// TwinCAT 3 PLC project Untitled1
// ProgramVersion: 3.1.4023.0
// libraries:
//   EfficientIO Communicator, * (EfficientIO)
//   EfficientIO Energy Basic, * (EfficientIO)
//   EfficientIO ModbusTCP, * (EfficientIO)
//   Lynus HTTP Functions, * (Lynus AG)
//   Lynus Standards, * (EfficientIO)
//   Tc2_Standard, * (Beckhoff Automation GmbH)
//   Tc2_System, * (Beckhoff Automation GmbH)
//   Tc2_Utilities, * (Beckhoff Automation GmbH)
//   Tc3_Module, * (Beckhoff Automation GmbH)
// project tree:
//   / Com.TcTTO, Lynus.TcTTO, PlcTask.TcTTO
//   DUTs/ struct_ADS_Auhofcenter.TcDUT
//   FBs/ FB_SPOpt_Monitoring_extTime.TcPOU
//   POUs/ MAIN.TcPOU, prgCom.TcPOU, prgLynus.TcPOU, prgPV.TcPOU
// real-time tasks:
//   TASK PlcTask: cycle T#10ms, priority 10, ADS port 350
//   TASK Com: cycle T#20ms, priority 14, ADS port 352
//   TASK Lynus: cycle T#5ms, priority 6, ADS port 351
//   TASK Riverside_Fast: cycle T#5ms, priority 8, ADS port 353
//   TASK Riverside_Middle: cycle T#20ms, priority 12, ADS port 354

CONFIGURATION Untitled1
    RESOURCE PLC ON TwinCAT3
        TASK Com(INTERVAL := T#20ms, PRIORITY := 14);
        TASK Lynus(INTERVAL := T#5ms, PRIORITY := 6);
        TASK PlcTask(INTERVAL := T#10ms, PRIORITY := 10);
        PROGRAM prgCom WITH Com : prgCom;
        PROGRAM prgLynus WITH Lynus : prgLynus;
        PROGRAM MAIN WITH PlcTask : MAIN;
        PROGRAM prgPV WITH PlcTask : prgPV;
    END_RESOURCE
END_CONFIGURATION

// ---- DUTs/struct_ADS_Auhofcenter.TcDUT
TYPE struct_ADS_Auhofcenter :
STRUCT
	int_liveCount		: INT;	
	rHeartbeat			: REAL;
	rErrorWarning		: REAL;
	rSPOptReady			: REAL;
	rUmfVorlaufSek		: REAL;
	rUmfRuecklaufSek	: REAL;
	bPumpenState		: BOOL;
	rRTMall_EG_Billa	: REAL;
	rRTMall_EG_RichutngBT2 : REAL;
	rRTMall_EG_VorPost 	: REAL;
	rRTMall_OG_Nordseitig : REAL;
	rRTMall_OG_Suedseitig : REAL;
	rRTMall_OG_VorTKMaxx : REAL;
	rRTMall_OG_VorStrasslSchaider : REAL;
	rNewTargetValue 	: REAL;
	rBT2UmfVorlaufSek	: REAL;
	rBT2UmfRuecklaufPri	: REAL;
	bBT2PumpenState		: BOOL;
	rBT2RTMall_EG_Nord	: REAL;
	rBT2RTMall_OG_Nord	: REAL;
	rBT2RTMall_EG_Sued	: REAL;
	rBT2RTMall_OG_Sued	: REAL;
	rBT2NewTargetValue	: REAL;
	rBT3UmfVorlaufSek	: REAL;
	rBT3UmfRuecklaufSek : REAL;
	bBT3PumpenState		: BOOL;
	rBT3RTMall_EG_West	: REAL;
	rBT3RTMall_OG_West	: REAL;
	rBT3RTMall_EG_HK31	: REAL;
	rBT3RTMall_EG_HK32	: REAL;
	rBT3RTMall_OG_K33	: REAL;
	rBT3RTMall_OG_K34	: REAL;
	rBT3RTMall_OG_Ost	: REAL;
	rBT3RTMall_EG_Ost	: REAL;
	rBT3RTMall_EG_HK35	: REAL;
	rBT3RTMall_OG_HK37	: REAL;
	rBT3NewTargetValue	: REAL;
	rBT4UmfVorlaufSek	: REAL;
	rBT4UmfRuecklaufSek	: REAL;
	bBT4PumpenState		: BOOL;
	rBT4RTMall_EG		: REAL;
	rBT5RTMall_OG		: REAL;
	rBT6RTMall_OG		: REAL;
	rBT6RTMall_EG		: REAL;
	rBT4NewTargetValue	: REAL;
	rAussentemperatur	: REAL;
	bEnableOp			: BOOL;
	bsEnableOp			: BOOL;
	bEnableOpBT2		: BOOL;
	bsEnableOpBT2		: BOOL;
	bEnableOpBT3		: BOOL;
	bsEnableOpBT3		: BOOL;
	bEnableOpBT4		: BOOL;
	bsEnableOpBT4		: BOOL;
	rBT1EM_Power_kW		: REAL;
	lrBT1EM_Counter_kWh	: REAL;
	rBT2EM_Power_kW		: REAL;
	lrBT2EM_Counter_kWh	: REAL;
	rBT3EM_Power_kW		: REAL;
	lrBT3EM_Counter_kWh	: REAL;
	rBT4EM_Power_kW		: REAL;
	lrBT4EM_Counter_kWh	: REAL;
	lrPowerPV_1_1		: LREAL;				
	lrPowerPV_1_2		: LREAL;				
	lrPowerPV_2_1		: LREAL;				
	lrPowerPV_2_2		: LREAL;				
	lrPowerPV_3_1		: LREAL;				
	lrPowerPV_3_2		: LREAL;				
	lrPowerPV_3_3		: LREAL;				
	lrPowerPV_3_4		: LREAL;				
	lrPowerPV_3_5		: LREAL;				
	lrPowerPV_3_6		: LREAL;				
	lrPowerPV			: LREAL;
	rUmfVorlaufPri		: REAL;
	rUmfRuecklaufPri	: REAL;
	rBT3UmfRuecklaufPri	: REAL;			
	rBT3UmfVorlaufPri	: REAL;
	rBT4UmfVorlaufPri	: REAL;
	rBT4UmfRuecklaufPri	: REAL;			
			(*: REAL;			
			: REAL;
			: REAL;			
			: REAL;			
			: REAL;
			: REAL;			
			: REAL;
			: REAL;			
*)

END_STRUCT
END_TYPE

// ---- POUs/prgCom.TcPOU
PROGRAM prgCom
VAR
	fbCom			: FB_MqttCommunicator_V5;
	byte_array : ARRAY[0..1023] OF BYTE;
	struct_transfer	: struct_ADS_Auhofcenter;
	mSize_to_Big: BOOL;
	uint_size: UINT;
END_VAR

fbCom(
	bConnect:= TRUE, 
	strAuthKey:=  'ENE87365342998' ,
	sUserName:= 'b605f16a-2d1c-4a4a-9b62-708dc1c64276', 
	sUserPassword:= 'e24298df-d4f0-45e5-b7c4-7373314a25dc', 
	eSavePositionCertificate:= eSavePositionOnPLC.ePostionC, 
	time_HeartBeat_sec := T#1S,
	bConnected=> , 
	bError=> , 
	hrErrorCode=> , 
	eConnectionState=> , 
	eErrorMessage_Out=> );
	
// copy values to struct	
struct_transfer.int_liveCount 				:= struct_transfer.int_liveCount+1;
struct_transfer.rHeartbeat			:= MAIN.rHeartbeat ;
struct_transfer.rErrorWarning		:= MAIN.rErrorWarning ;
struct_transfer.rSPOptReady			:= MAIN.rSPOptReady ;
struct_transfer.rUmfVorlaufSek		:= MAIN.rUmfVorlaufSek ;
struct_transfer.rUmfRuecklaufSek	:=  MAIN.rUmfRuecklaufSek;
struct_transfer.bPumpenState		:= MAIN.bPumpenState ;
struct_transfer.rRTMall_EG_Billa	:= MAIN.rRTMall_EG_Billa ;
struct_transfer.rRTMall_EG_RichutngBT2	:= MAIN.rRTMall_EG_RichutngBT2 ;
struct_transfer.rRTMall_EG_VorPost	:=  MAIN.rRTMall_EG_VorPost;
struct_transfer.rRTMall_OG_Nordseitig :=  MAIN.rRTMall_OG_Nordseitig;
struct_transfer.rRTMall_OG_Suedseitig := MAIN.rRTMall_OG_Suedseitig ;
struct_transfer.rRTMall_OG_VorTKMaxx := MAIN.rRTMall_OG_VorTKMaxx ;
struct_transfer.rRTMall_OG_VorStrasslSchaider :=  MAIN.rRTMall_OG_VorStrasslSchaider;
struct_transfer.rNewTargetValue		:= MAIN.rNewTargetValue ;
struct_transfer.rBT2UmfVorlaufSek	:= MAIN.rBT2UmfVorlaufSek ;
struct_transfer.rBT2UmfRuecklaufPri	:= MAIN.rBT2UmfRuecklaufPri ;
struct_transfer.bBT2PumpenState		:=  MAIN.bBT2PumpenState;
struct_transfer.rBT2RTMall_EG_Nord	:= MAIN.rBT2RTMall_EG_Nord ;
struct_transfer.rBT2RTMall_OG_Nord	:= MAIN.rBT2RTMall_OG_Nord ;
struct_transfer.rBT2RTMall_EG_Sued	:= MAIN.rBT2RTMall_EG_Sued ;
struct_transfer.rBT2RTMall_OG_Sued	:= MAIN.rBT2RTMall_OG_Sued ;
struct_transfer.rBT2NewTargetValue	:= MAIN.rBT2NewTargetValue ;
struct_transfer.rBT3UmfVorlaufSek	:= MAIN.rBT3UmfVorlaufSek ;
struct_transfer.rBT3UmfRuecklaufSek	:= MAIN.rBT3UmfRuecklaufSek ;
struct_transfer.bBT3PumpenState		:= MAIN.bBT3PumpenState ;
struct_transfer.rBT3RTMall_EG_West	:= MAIN.rBT3RTMall_EG_West ;
struct_transfer.rBT3RTMall_OG_West	:= MAIN.rBT3RTMall_OG_West ;
struct_transfer.rBT3RTMall_EG_HK31	:= MAIN.rBT3RTMall_EG_HK31 ;
struct_transfer.rBT3RTMall_EG_HK32	:= MAIN.rBT3RTMall_EG_HK32 ;
struct_transfer.rBT3RTMall_OG_K33	:= MAIN.rBT3RTMall_OG_K33 ;
struct_transfer.rBT3RTMall_OG_K34	:= MAIN.rBT3RTMall_OG_K34 ;
struct_transfer.rBT3RTMall_OG_Ost	:= MAIN.rBT3RTMall_OG_Ost ;
struct_transfer.rBT3RTMall_EG_Ost	:=  MAIN.rBT3RTMall_EG_Ost;
struct_transfer.rBT3RTMall_EG_HK35	:= MAIN.rBT3RTMall_EG_HK35 ;
struct_transfer.rBT3RTMall_OG_HK37	:= MAIN.rBT3RTMall_OG_HK37 ;
struct_transfer.rBT3NewTargetValue	:= MAIN.rBT3NewTargetValue ;
struct_transfer.rBT4UmfVorlaufSek	:= MAIN.rBT4UmfVorlaufSek ;
struct_transfer.rBT4UmfRuecklaufSek	:= MAIN.rBT4UmfRuecklaufSek ;
struct_transfer.bBT4PumpenState		:= MAIN.bBT4PumpenState ;
struct_transfer.rBT4RTMall_EG		:= MAIN.rBT4RTMall_EG ;
struct_transfer.rBT5RTMall_OG		:= MAIN.rBT5RTMall_OG ;
struct_transfer.rBT6RTMall_OG		:= MAIN.rBT6RTMall_OG ;
struct_transfer.rBT6RTMall_EG		:= MAIN.rBT6RTMall_EG ;
struct_transfer.rBT4NewTargetValue	:= MAIN.rBT4NewTargetValue ;
struct_transfer.rAussentemperatur	:= MAIN.rAussentemperatur ;
struct_transfer.bEnableOp			:= MAIN.bEnableOp ;
struct_transfer.bSEnableOp			:= MAIN.bSEnableOp ;
struct_transfer.bEnableOpBT2		:= MAIN.bEnableOpBT2 ;
struct_transfer.bSEnableOpBT2		:= MAIN.bSEnableOpBT2 ;
struct_transfer.bEnableOpBT3		:= MAIN.bEnableOpBT3 ;
struct_transfer.bSEnableOpBT3		:= MAIN.bSEnableOpBT3 ;
struct_transfer.bEnableOpBT4		:= MAIN.bEnableOpBT4 ;
struct_transfer.bSEnableOpBT4		:= MAIN.bSEnableOpBT4 ;
struct_transfer.rBT1EM_Power_kW		:= MAIN.rBT1EM_Power_kW ;
struct_transfer.lrBT1EM_Counter_kWh	:= MAIN.lrBT1EM_Counter_kWh ;
struct_transfer.rBT2EM_Power_kW		:= MAIN.rBT2EM_Power_kW ;
struct_transfer.lrBT2EM_Counter_kWh	:= MAIN.lrBT2EM_Counter_kWh ;
struct_transfer.rBT3EM_Power_kW		:= MAIN.rBT3EM_Power_kW ;
struct_transfer.lrBT3EM_Counter_kWh	:= MAIN.lrBT3EM_Counter_kWh ;
struct_transfer.rBT4EM_Power_kW		:= MAIN.rBT4EM_Power_kW ;
struct_transfer.lrBT4EM_Counter_kWh	:= MAIN.lrBT4EM_Counter_kWh ;
struct_transfer.lrPowerPV_1_1		:= prgPV.lrPowerPV_1_1 ;
struct_transfer.lrPowerPV_1_2		:= prgPV.lrPowerPV_1_2 ;
struct_transfer.lrPowerPV_2_1		:= prgPV.lrPowerPV_2_1 ;
struct_transfer.lrPowerPV_2_2		:= prgPV.lrPowerPV_2_2 ;
struct_transfer.lrPowerPV_3_1		:= prgPV.lrPowerPV_3_1 ;
struct_transfer.lrPowerPV_3_2		:= prgPV.lrPowerPV_3_2 ;
struct_transfer.lrPowerPV_3_3		:= prgPV.lrPowerPV_3_3 ;
struct_transfer.lrPowerPV_3_4		:= prgPV.lrPowerPV_3_4 ;
struct_transfer.lrPowerPV_3_5		:= prgPV.lrPowerPV_3_5 ;
struct_transfer.lrPowerPV_3_6		:= prgPV.lrPowerPV_3_6 ;
struct_transfer.lrPowerPV			:= prgPV.lrPowerPV ;
struct_transfer.rUmfVorlaufPri		:=  MAIN.rUmfVorlaufPri;
struct_transfer.rUmfRuecklaufPri	:=  Main.rUmfRuecklaufPri;
struct_transfer.rBT3UmfRuecklaufPri		:= MAIN.rBT3UmfRuecklaufPri ;
struct_transfer.rBT3UmfVorlaufPri		:= MAIN.rBT3UmfVorlaufPri ;
struct_transfer.rBT4UmfVorlaufPri		:=  Main.rBT4UmfVorlaufPri;
struct_transfer.rBT4UmfRuecklaufPri		:= MAIN.rBT4UmfRuecklaufPri ;
(*struct_transfer.		:=  ;
struct_transfer.		:=  ;
struct_transfer.		:=  ;
struct_transfer.		:=  ;
struct_transfer.		:=  ;
struct_transfer.		:=  ;
*)

// copy struct to byte array
IF SIZEOF(struct_transfer) > SIZEOF(byte_array) THEN
	memcpy(ADR(byte_array),ADR(struct_transfer),SIZEOF(byte_array));
	uint_size := SIZEOF(struct_transfer);
	mSize_to_Big := TRUE;
ELSE
	memcpy(ADR(byte_array),ADR(struct_transfer),SIZEOF(struct_transfer));
	mSize_to_Big := FALSE;
END_IF
uint_size := SIZEOF(struct_transfer);

END_PROGRAM

// ---- POUs/MAIN.TcPOU
PROGRAM MAIN
VAR
	fbVarInfo						: FB_VarInfo;	
	timStart						: TON;
	timResetConnection				: TON;
	byLPArr							: BYTE;
	iState							: INT;	
	uiErrorCounter					: UINT;
	rHeartbeat						: REAL;			//{#lynus.ag#()}
	rErrorWarning					: REAL;			//{#lynus.ag#()}
	rSPOptReady						: REAL;			//{#lynus.ag#()}
	FPStart							: R_TRIG;
	FPDone							: R_TRIG;
	FPError							: R_TRIG;
	fbHttp							: FB_GetSet_Data_Auhofcenter;
		
	// Bauteil1
	fbMonitor						: FB_SPOpt_Monitoring_extTime;
	bSEnableOp						: BOOL;			//{#lynus.ag#()}
	byHB							: BYTE;			//Watchdog
	rNewTargetValue					: REAL;			//{#lynus.ag#()} //Optimierter Sollwert Vorlauftemperatur
	bPumpenState					: BOOL;			//{#lynus.ag#()} //Heizung Aus/Ein (Hauptschalter)
	rAussentemperatur				: REAL;			//{#lynus.ag#()} //Aussentemperatur 
	rUmfVorlaufPri					: REAL;			//{#lynus.ag#()} //Umformer Vorlauftemperatur primär
	rUmfRuecklaufPri				: REAL;			//{#lynus.ag#()} //Umformer Rücklauftemperatur primär
	rUmfVorlaufSek					: REAL;			//{#lynus.ag#()} //Umformer Vorlauftemperatur sekundär
	rUmfRuecklaufSek				: REAL;			//{#lynus.ag#()} //Umformer Rücklauftemperatur sekundär
	rRTMall_EG_Billa				: REAL;			//{#lynus.ag#()} //Raumtemperatur Mall EG, vor Billa
	rRTMall_EG_RichutngBT2			: REAL;			//{#lynus.ag#()} //Raumtemperatur Mall EG, Richtung Bauteil 2
	rRTMall_EG_VorPost				: REAL;			//{#lynus.ag#()} //Raumtemperatur Mall EG, vor Post
	rRTMall_OG_VorTKMaxx			: REAL;			//{#lynus.ag#()} //Raumtemperatur Mall 1. OG, vor TKMaxx
	rRTMall_OG_VorStrasslSchaider	: REAL;			//{#lynus.ag#()} //Raumtemperatur Mall 1. OG, vor Strassl-Schaider
	rRTMall_OG_Nordseitig			: REAL;			//{#lynus.ag#()} //Raumtemperatur Mall 2. OG, Nordseitig
	rRTMall_OG_Suedseitig			: REAL;			//{#lynus.ag#()} //Raumtemperatur Mall 2. OG, Südseitig
	
	// Bauteil2
	fbMonitorBT2					: FB_SPOpt_Monitoring_extTime;
	bSEnableOpBT2					: BOOL;			//{#lynus.ag#()}
	byBT2HB							: BYTE;			//Watchdog
	bBT2PumpenState					: BOOL;			//{#lynus.ag#()} //Heizung Aus/Ein (Hauptschalter)
	rBT2NewTargetValue				: REAL;			//{#lynus.ag#()} //Optimierter Sollwert Vorlauftemperatur
	rBT2UmfVorlaufSek				: REAL;			//{#lynus.ag#()} //Umformer Vorlauftemperatur sekundär
	rBT2UmfRuecklaufPri				: REAL;			//{#lynus.ag#()} //Umformer Rücklauftemperatur primär
	rBT2RTMall_EG_Nord				: REAL;			//{#lynus.ag#()} //Raumtemperatur Mall EG, Nord
	rBT2RTMall_OG_Nord				: REAL;			//{#lynus.ag#()} //Raumtemperatur Mall OG, Nord
	rBT2RTMall_EG_Sued				: REAL;			//{#lynus.ag#()} //Raumtemperatur Mall EG, Sued
	rBT2RTMall_OG_Sued				: REAL;			//{#lynus.ag#()} //Raumtemperatur Mall OG, Sued
	
	// Bauteil3
	fbMonitorBT3					: FB_SPOpt_Monitoring_extTime;
	bSEnableOpBT3					: BOOL;			//{#lynus.ag#()}
	byBT3HB							: BYTE;			//Watchdog
	bBT3PumpenState					: BOOL;			//{#lynus.ag#()} //Heizung Aus/Ein (Hauptschalter)
	rBT3NewTargetValue				: REAL;			//{#lynus.ag#()} //Optimierter Sollwert Vorlauftemperatur
	rBT3UmfVorlaufPri				: REAL;			//{#lynus.ag#()} //Umformer Vorlauftemperatur primär
	rBT3UmfRuecklaufPri				: REAL;			//{#lynus.ag#()} //Umformer Rücklauftemperatur primär
	rBT3UmfVorlaufSek				: REAL;			//{#lynus.ag#()} //Umformer Vorlauftemperatur sekundär
	rBT3UmfRuecklaufSek				: REAL;			//{#lynus.ag#()} //Umformer Rücklauftemperatur sekundär
	rBT3RTMall_EG_West				: REAL;			//{#lynus.ag#()} //Raumtemperatur Mall EG, West
	rBT3RTMall_OG_West				: REAL;			//{#lynus.ag#()} //Raumtemperatur Mall OG, West
	rBT3RTMall_EG_HK31				: REAL;			//{#lynus.ag#()} //Raumtemperatur Mall EG, HK3.1
	rBT3RTMall_EG_HK32				: REAL;			//{#lynus.ag#()} //Raumtemperatur Mall EG, HK3.2
	rBT3RTMall_OG_K33				: REAL;			//{#lynus.ag#()} //Raumtemperatur Mall OG, K3.3
	rBT3RTMall_OG_K34				: REAL;			//{#lynus.ag#()} //Raumtemperatur Mall OG, K3.4
	rBT3RTMall_OG_Ost				: REAL;			//{#lynus.ag#()} //Raumtemperatur Mall OG, Ost
	rBT3RTMall_EG_Ost				: REAL;			//{#lynus.ag#()} //Raumtemperatur Mall EG, Ost
	rBT3RTMall_EG_HK35				: REAL;			//{#lynus.ag#()} //Raumtemperatur Mall EG, HK3.5
	rBT3RTMall_OG_HK37				: REAL;			//{#lynus.ag#()} //Raumtemperatur Mall OG, HK3.7
	
	// Bauteil4
	fbMonitorBT4					: FB_SPOpt_Monitoring_extTime;
	bSEnableOpBT4					: BOOL;			//{#lynus.ag#()}
	byBT4HB							: BYTE;			//Watchdog
	bBT4PumpenState					: BOOL;			//{#lynus.ag#()} //Heizung Aus/Ein (Hauptschalter)
	rBT4NewTargetValue				: REAL;			//{#lynus.ag#()} //Optimierter Sollwert Vorlauftemperatur
	rBT4UmfVorlaufPri				: REAL;			//{#lynus.ag#()} //Umformer Vorlauftemperatur primär
	rBT4UmfRuecklaufPri				: REAL;			//{#lynus.ag#()} //Umformer Rücklauftemperatur primär
	rBT4UmfVorlaufSek				: REAL;			//{#lynus.ag#()} //Umformer Vorlauftemperatur sekundär
	rBT4UmfRuecklaufSek				: REAL;			//{#lynus.ag#()} //Umformer Rücklauftemperatur sekundär
	rBT4RTMall_EG					: REAL;			//{#lynus.ag#()} //Raumtemperatur Mall EG
	rBT5RTMall_OG					: REAL;			//{#lynus.ag#()} //Raumtemperatur Mall OG (BT5)
	rBT6RTMall_OG					: REAL;			//{#lynus.ag#()} //Raumtemperatur Mall OG (BT6)
	rBT6RTMall_EG					: REAL;			//{#lynus.ag#()} //Raumtemperatur Mall EG (BT6)

	// Wurzelzaehler
	lrBT1EM_Counter_kWh				: LREAL;		//{#lynus.ag#()} //BT1 Zaehlerstand	
	rBT1EM_Power_kW					: REAL;			//{#lynus.ag#()} //BT1 Momentanleistung
	lrBT2EM_Counter_kWh				: LREAL;		//{#lynus.ag#()} //BT2 Zaehlerstand
	rBT2EM_Power_kW					: REAL;			//{#lynus.ag#()} //BT2 Momentanleistung
	lrBT3EM_Counter_kWh				: LREAL;		//{#lynus.ag#()} //BT3 Zaehlerstand
	rBT3EM_Power_kW					: REAL;			//{#lynus.ag#()} //BT3 Momentanleistung
	lrBT4EM_Counter_kWh				: LREAL;		//{#lynus.ag#()} //BT4 Zaehlerstand
	rBT4EM_Power_kW					: REAL;			//{#lynus.ag#()} //BT4 Momentanleistung

	x: INT;
	
	bDissableExtHBBT1 : BOOL;			//{#lynus.ag#()}
	bDissableExtHBBT2 : BOOL;			//{#lynus.ag#()}
	bDissableExtHBBT3 : BOOL;			//{#lynus.ag#()}
	bDissableExtHBBT4 : BOOL;			//{#lynus.ag#()}

END_VAR
VAR PERSISTENT
	bEnableOp						: BOOL;			//{#lynus.ag#()}
	bEnableOpBT2					: BOOL;			//{#lynus.ag#()}
	bEnableOpBT3					: BOOL;			//{#lynus.ag#()}
	bEnableOpBT4					: BOOL;			//{#lynus.ag#()}
END_VAR

//Search the Variabels for Lynus
fbVarInfo(
	bReadInfo:= , 
	eTMCFile:= eSelectTMCFile.eDontUseTMCFile, 
	eSavePositionTMCFile:= eSavePositionOnPLC.ePostionC, 
	udiCounterFoundVariables=> , 
	bError=> , 
	bBusy=> , 
	byProgress=> , 
	udiErrorCodeOut=> , 
	eErrorVarInfo_Out=> , 
	sVarWithError=> );

//Monitor
fbMonitor(
	bEnable:= bEnableOp, 
	bDissableHB:= FALSE, 
	tChangeHBIn:= T#1H, 
	tChangeHBOut:= T#30S, 
	rHeartbeat:= rHeartbeat, 
	rErrorWarning:= rErrorWarning, 
	rSPOptReady:= rSPOptReady,
	bReadyOut=> , 
	bDissableExtHB=> bDissableExtHBBT1, 
	bSEnable=> bSEnableOp, 
	rHeartbeatOut=> );

//Monitor BT2
fbMonitorBT2(
	bEnable:= bEnableOpBT2, 
	bDissableHB:= FALSE, 
	tChangeHBIn:= T#1H, 
	tChangeHBOut:= T#30S, 
	rHeartbeat:= rHeartbeat, 
	rErrorWarning:= rErrorWarning, 
	rSPOptReady:= rSPOptReady,
	bReadyOut=> , 
	bDissableExtHB=> bDissableExtHBBT2, 
	bSEnable=> bSEnableOpBT2, 
	rHeartbeatOut=> );
	
//Monitor BT3
fbMonitorBT3(
	bEnable:= bEnableOpBT3, 
	bDissableHB:= FALSE, 
	tChangeHBIn:= T#1H, 
	tChangeHBOut:= T#30S, 
	rHeartbeat:= rHeartbeat, 
	rErrorWarning:= rErrorWarning, 
	rSPOptReady:= rSPOptReady,
	bReadyOut=> , 
	bDissableExtHB=> bDissableExtHBBT3, 
	bSEnable=> bSEnableOpBT3, 
	rHeartbeatOut=> );
	
//Monitor BT4
fbMonitorBT4(
	bEnable:= bEnableOpBT4, 
	bDissableHB:= FALSE, 
	tChangeHBIn:= T#1H, 
	tChangeHBOut:= T#30S, 
	rHeartbeat:= rHeartbeat, 
	rErrorWarning:= rErrorWarning, 
	rSPOptReady:= rSPOptReady,
	bReadyOut=> , 
	bDissableExtHB=> bDissableExtHBBT4, 
	bSEnable=> bSEnableOpBT4, 
	rHeartbeatOut=> );
	
//Read/Write Function to the Auhofcenter System	
timStart(IN:= TRUE, PT:= T#5S, Q=> , ET=> );

FPStart(CLK:= timStart.Q, Q=> );

IF FPStart.Q THEN
	iState := 1;	
END_IF

CASE iState OF

	0://Stop
		fbHttp.bStart := FALSE;

	1://Read Values
		fbHttp.bStart := TRUE;	
			fbHttp.bReadRequest := TRUE;
				fbHttp.bWriteRequest := FALSE;
		
		(* ----- Variablen Bauteil 1 ----- *)
		//Aussentemperatur (Mittelwert aus 4 Messstellen)	
		fbHttp.arrListOfVariables[1].bIsString := FALSE;
			fbHttp.arrListOfVariables[1].sVariableName := 'DV100';	
				fbHttp.arrListOfVariables[1].sVariableValue := '';	
		//Umformer Vorlauftemperatur primär
		fbHttp.arrListOfVariables[2].bIsString := FALSE;
			fbHttp.arrListOfVariables[2].sVariableName := 'DV111';
				fbHttp.arrListOfVariables[2].sVariableValue := '';	
		//Umformer Rücklauftemperatur primär
		fbHttp.arrListOfVariables[3].bIsString := FALSE;
			fbHttp.arrListOfVariables[3].sVariableName := 'DV112';
				fbHttp.arrListOfVariables[3].sVariableValue := '';
		//Umformer Vorlauftemperatur sekundär
		fbHttp.arrListOfVariables[4].bIsString := FALSE;
			fbHttp.arrListOfVariables[4].sVariableName := 'DV113';
				fbHttp.arrListOfVariables[4].sVariableValue := '';
		//Umformer Rücklauftemperatur sekundär
		fbHttp.arrListOfVariables[5].bIsString := FALSE;
			fbHttp.arrListOfVariables[5].sVariableName := 'DV114';
				fbHttp.arrListOfVariables[5].sVariableValue := '';	
		//Raumtemperatur Mall EG, vor Billa
		fbHttp.arrListOfVariables[6].bIsString := FALSE;
			fbHttp.arrListOfVariables[6].sVariableName := 'DV121';
				fbHttp.arrListOfVariables[6].sVariableValue := '';
		//Raumtemperatur Mall EG, Richtung BT2
		fbHttp.arrListOfVariables[7].bIsString := FALSE;
			fbHttp.arrListOfVariables[7].sVariableName := 'DV122';
				fbHttp.arrListOfVariables[7].sVariableValue := '';
		//Raumtemperatur Mall EG, vor Post
		fbHttp.arrListOfVariables[8].bIsString := FALSE;
			fbHttp.arrListOfVariables[8].sVariableName := 'DV123';
				fbHttp.arrListOfVariables[8].sVariableValue := '';
		//Raumtemperatur Mall 1. OG, vor TKMaxx
		fbHttp.arrListOfVariables[9].bIsString := FALSE;
			fbHttp.arrListOfVariables[9].sVariableName := 'DV124';
				fbHttp.arrListOfVariables[9].sVariableValue := '';
		//Raumtemperatur Mall 1. OG, vor Strassl-Schaider
		fbHttp.arrListOfVariables[10].bIsString := FALSE;
			fbHttp.arrListOfVariables[10].sVariableName := 'DV125';
				fbHttp.arrListOfVariables[10].sVariableValue := '';
		//Raumtemperatur Mall 2. OG, Nordseitig
		fbHttp.arrListOfVariables[11].bIsString := FALSE;
			fbHttp.arrListOfVariables[11].sVariableName := 'DV126';
				fbHttp.arrListOfVariables[11].sVariableValue := '';
		//Raumtemperatur Mall 2. OG, Südseitig
		fbHttp.arrListOfVariables[12].bIsString := FALSE;
			fbHttp.arrListOfVariables[12].sVariableName := 'DV127';
				fbHttp.arrListOfVariables[12].sVariableValue := '';
		//Status Pumpe
		fbHttp.arrListOfVariables[13].bIsString := FALSE;
			fbHttp.arrListOfVariables[13].sVariableName := 'DV128';
				fbHttp.arrListOfVariables[13].sVariableValue := '';
		
		(* ----- Variablen Bauteil 2 ----- *)
		//Umformer Vorlauftemperatur sekundär	
		fbHttp.arrListOfVariables[14].bIsString := FALSE;
			fbHttp.arrListOfVariables[14].sVariableName := 'DV211';	
				fbHttp.arrListOfVariables[14].sVariableValue := '';
		//Umformer Rücklauftemperatur primär
		fbHttp.arrListOfVariables[15].bIsString := FALSE;
			fbHttp.arrListOfVariables[15].sVariableName := 'DV212';	
				fbHttp.arrListOfVariables[15].sVariableValue := '';
		//Raumtemperatur Mall EG, Nord
		fbHttp.arrListOfVariables[16].bIsString := FALSE;
			fbHttp.arrListOfVariables[16].sVariableName := 'DV221';	
				fbHttp.arrListOfVariables[16].sVariableValue := '';
		//Raumtemperatur Mall OG, Nord
		fbHttp.arrListOfVariables[17].bIsString := FALSE;
			fbHttp.arrListOfVariables[17].sVariableName := 'DV222';	
				fbHttp.arrListOfVariables[17].sVariableValue := '';
		//Raumtemperatur Mall EG, Süd
		fbHttp.arrListOfVariables[18].bIsString := FALSE;
			fbHttp.arrListOfVariables[18].sVariableName := 'DV223';	
				fbHttp.arrListOfVariables[18].sVariableValue := '';
		//Raumtemperatur Mall OG, Süd
		fbHttp.arrListOfVariables[19].bIsString := FALSE;
			fbHttp.arrListOfVariables[19].sVariableName := 'DV224';	
				fbHttp.arrListOfVariables[19].sVariableValue := '';
		//Heizung Aus/Ein (Hauptschalter)
		fbHttp.arrListOfVariables[20].bIsString := FALSE;
			fbHttp.arrListOfVariables[20].sVariableName := 'DV232';	
				fbHttp.arrListOfVariables[20].sVariableValue := '';
				
		(* ----- Variablen Bauteil 3 ----- *)
		//Umformer Vorlauftemperatur primär	
		fbHttp.arrListOfVariables[21].bIsString := FALSE;
			fbHttp.arrListOfVariables[21].sVariableName := 'DV311';	
				fbHttp.arrListOfVariables[21].sVariableValue := '';
		//Umformer Rücklauftemperatur primär
		fbHttp.arrListOfVariables[22].bIsString := FALSE;
			fbHttp.arrListOfVariables[22].sVariableName := 'DV312';	
				fbHttp.arrListOfVariables[22].sVariableValue := '';
		//Umformer Vorlauftemperatur sekundär
		fbHttp.arrListOfVariables[23].bIsString := FALSE;
			fbHttp.arrListOfVariables[23].sVariableName := 'DV313';	
				fbHttp.arrListOfVariables[23].sVariableValue := '';
		//Umformer Rücklauftemperatur sekundär
		fbHttp.arrListOfVariables[24].bIsString := FALSE;
			fbHttp.arrListOfVariables[24].sVariableName := 'DV314';	
				fbHttp.arrListOfVariables[24].sVariableValue := '';
		//Raumtemperatur Mall EG, West
		fbHttp.arrListOfVariables[25].bIsString := FALSE;
			fbHttp.arrListOfVariables[25].sVariableName := 'DV321';	
				fbHttp.arrListOfVariables[25].sVariableValue := '';
		//Raumtemperatur Mall OG, West
		fbHttp.arrListOfVariables[26].bIsString := FALSE;
			fbHttp.arrListOfVariables[26].sVariableName := 'DV322';	
				fbHttp.arrListOfVariables[26].sVariableValue := '';
		//Raumtemperatur Mall EG (HK3.1)
		fbHttp.arrListOfVariables[27].bIsString := FALSE;
			fbHttp.arrListOfVariables[27].sVariableName := 'DV323';	
				fbHttp.arrListOfVariables[27].sVariableValue := '';
		//Raumtemperatur Mall EG (HK3.2)
		fbHttp.arrListOfVariables[28].bIsString := FALSE;
			fbHttp.arrListOfVariables[28].sVariableName := 'DV324';	
				fbHttp.arrListOfVariables[28].sVariableValue := '';
		//Raumtemperatur Mall OG (K3.3)
		fbHttp.arrListOfVariables[29].bIsString := FALSE;
			fbHttp.arrListOfVariables[29].sVariableName := 'DV325';	
				fbHttp.arrListOfVariables[29].sVariableValue := '';
		//Raumtemperatur Mall OG (K3.4)
		fbHttp.arrListOfVariables[30].bIsString := FALSE;
			fbHttp.arrListOfVariables[30].sVariableName := 'DV326';	
				fbHttp.arrListOfVariables[30].sVariableValue := '';
		//Raumtemperatur Mall OG, Ost
		fbHttp.arrListOfVariables[31].bIsString := FALSE;
			fbHttp.arrListOfVariables[31].sVariableName := 'DV327';	
				fbHttp.arrListOfVariables[31].sVariableValue := '';
		//Raumtemperatur Mall EG, Ost
		fbHttp.arrListOfVariables[32].bIsString := FALSE;
			fbHttp.arrListOfVariables[32].sVariableName := 'DV328';	
				fbHttp.arrListOfVariables[32].sVariableValue := '';
		//Raumtemperatur Mall EG (HK3.5)
		fbHttp.arrListOfVariables[33].bIsString := FALSE;
			fbHttp.arrListOfVariables[33].sVariableName := 'DV329';	
				fbHttp.arrListOfVariables[33].sVariableValue := '';
		//Raumtemperatur Mall OG (K3.7)
		fbHttp.arrListOfVariables[34].bIsString := FALSE;
			fbHttp.arrListOfVariables[34].sVariableName := 'DV330';	
				fbHttp.arrListOfVariables[34].sVariableValue := '';
		//Heizung Aus/Ein (Hauptschalter)
		fbHttp.arrListOfVariables[35].bIsString := FALSE;
			fbHttp.arrListOfVariables[35].sVariableName := 'DV333';	
				fbHttp.arrListOfVariables[35].sVariableValue := '';
		
		(* ----- Variablen Bauteil 4 ----- *)
		//Umformer Vorlauftemperatur primär
		fbHttp.arrListOfVariables[36].bIsString := FALSE;
			fbHttp.arrListOfVariables[36].sVariableName := 'DV411';	
				fbHttp.arrListOfVariables[36].sVariableValue := '';
		//Umformer Rücklauftemperatur primär
		fbHttp.arrListOfVariables[37].bIsString := FALSE;
			fbHttp.arrListOfVariables[37].sVariableName := 'DV412';	
				fbHttp.arrListOfVariables[37].sVariableValue := '';
		//Umformer Vorlauftemperatur sekundär
		fbHttp.arrListOfVariables[38].bIsString := FALSE;
			fbHttp.arrListOfVariables[38].sVariableName := 'DV413';	
				fbHttp.arrListOfVariables[38].sVariableValue := '';
		//Umformer Rücklauftemperatur sekundär
		fbHttp.arrListOfVariables[39].bIsString := FALSE;
			fbHttp.arrListOfVariables[39].sVariableName := 'DV414';	
				fbHttp.arrListOfVariables[39].sVariableValue := '';
		//Raumtemperatur Mall EG
		fbHttp.arrListOfVariables[40].bIsString := FALSE;
			fbHttp.arrListOfVariables[40].sVariableName := 'DV421';	
				fbHttp.arrListOfVariables[40].sVariableValue := '';
		//BT5 Raumtemperatur Mall OG
		fbHttp.arrListOfVariables[41].bIsString := FALSE;
			fbHttp.arrListOfVariables[41].sVariableName := 'DV422';	
				fbHttp.arrListOfVariables[41].sVariableValue := '';
		//BT6 Raumtemperatur Mall OG
		fbHttp.arrListOfVariables[42].bIsString := FALSE;
			fbHttp.arrListOfVariables[42].sVariableName := 'DV423';	
				fbHttp.arrListOfVariables[42].sVariableValue := '';
		//BT6 Raumtemperatur Mall EG
		fbHttp.arrListOfVariables[43].bIsString := FALSE;
			fbHttp.arrListOfVariables[43].sVariableName := 'DV424';	
				fbHttp.arrListOfVariables[43].sVariableValue := '';
		//Heizung Aus/Ein (Hauptschalter)
		fbHttp.arrListOfVariables[44].bIsString := FALSE;
			fbHttp.arrListOfVariables[44].sVariableName := 'DV432';	
				fbHttp.arrListOfVariables[44].sVariableValue := '';
		
		(* ----- Variablen Wurzelzaehler ----- *)
		//BT1 Zaehlerstand
		fbHttp.arrListOfVariables[45].bIsString := FALSE;
			fbHttp.arrListOfVariables[45].sVariableName := 'DV510';	
				fbHttp.arrListOfVariables[45].sVariableValue := '';
		//BT1 Momentanleistung
		fbHttp.arrListOfVariables[46].bIsString := FALSE;
			fbHttp.arrListOfVariables[46].sVariableName := 'DV511';	
				fbHttp.arrListOfVariables[46].sVariableValue := '';
		//BT2 Zaehlerstand
		fbHttp.arrListOfVariables[47].bIsString := FALSE;
			fbHttp.arrListOfVariables[47].sVariableName := 'DV520';	
				fbHttp.arrListOfVariables[47].sVariableValue := '';
		//BT2 Momentanleistung
		fbHttp.arrListOfVariables[48].bIsString := FALSE;
			fbHttp.arrListOfVariables[48].sVariableName := 'DV521';	
				fbHttp.arrListOfVariables[48].sVariableValue := '';
		//BT3 Zaehlerstand
		fbHttp.arrListOfVariables[49].bIsString := FALSE;
			fbHttp.arrListOfVariables[49].sVariableName := 'DV530';	
				fbHttp.arrListOfVariables[49].sVariableValue := '';
		//BT3 Momentanleistung
		fbHttp.arrListOfVariables[50].bIsString := FALSE;
			fbHttp.arrListOfVariables[50].sVariableName := 'DV531';	
				fbHttp.arrListOfVariables[50].sVariableValue := '';
		//BT4 Zaehlerstand
		fbHttp.arrListOfVariables[51].bIsString := FALSE;
			fbHttp.arrListOfVariables[51].sVariableName := 'DV540';	
				fbHttp.arrListOfVariables[51].sVariableValue := '';
		//BT4 Momentanleistung
		fbHttp.arrListOfVariables[52].bIsString := FALSE;
			fbHttp.arrListOfVariables[52].sVariableName := 'DV541';	
				fbHttp.arrListOfVariables[52].sVariableValue := '';

	
		IF FPDone.Q THEN 
			iState := 2; 
				//Auf Lynus Variablen mappen
				(* ----- Variablen Bauteil 1 ----- *)
				rAussentemperatur := STRING_TO_REAL(fbHttp.arrListOfVariabelsOut[1].sVariableValue);
				rUmfVorlaufPri := STRING_TO_REAL(fbHttp.arrListOfVariabelsOut[2].sVariableValue);
				rUmfRuecklaufPri := STRING_TO_REAL(fbHttp.arrListOfVariabelsOut[3].sVariableValue);
				rUmfVorlaufSek := STRING_TO_REAL(fbHttp.arrListOfVariabelsOut[4].sVariableValue);
				rUmfRuecklaufSek := STRING_TO_REAL(fbHttp.arrListOfVariabelsOut[5].sVariableValue);
				rRTMall_EG_Billa := STRING_TO_REAL(fbHttp.arrListOfVariabelsOut[6].sVariableValue);
				rRTMall_EG_RichutngBT2 := STRING_TO_REAL(fbHttp.arrListOfVariabelsOut[7].sVariableValue);
				rRTMall_EG_VorPost := STRING_TO_REAL(fbHttp.arrListOfVariabelsOut[8].sVariableValue);
				rRTMall_OG_VorTKMaxx := STRING_TO_REAL(fbHttp.arrListOfVariabelsOut[9].sVariableValue);
				rRTMall_OG_VorStrasslSchaider := STRING_TO_REAL(fbHttp.arrListOfVariabelsOut[10].sVariableValue);
				rRTMall_OG_Nordseitig := STRING_TO_REAL(fbHttp.arrListOfVariabelsOut[11].sVariableValue);
				rRTMall_OG_Suedseitig := STRING_TO_REAL(fbHttp.arrListOfVariabelsOut[12].sVariableValue);
				bPumpenState := DINT_TO_BOOL(STRING_TO_DINT(fbHttp.arrListOfVariabelsOut[13].sVariableValue));
				
				(* ----- Variablen Bauteil 2 ----- *)
				rBT2UmfVorlaufSek := STRING_TO_REAL(fbHttp.arrListOfVariabelsOut[14].sVariableValue);
				rBT2UmfRuecklaufPri := STRING_TO_REAL(fbHttp.arrListOfVariabelsOut[15].sVariableValue);
				rBT2RTMall_EG_Nord := STRING_TO_REAL(fbHttp.arrListOfVariabelsOut[16].sVariableValue);
				rBT2RTMall_OG_Nord := STRING_TO_REAL(fbHttp.arrListOfVariabelsOut[17].sVariableValue);
				rBT2RTMall_EG_Sued := STRING_TO_REAL(fbHttp.arrListOfVariabelsOut[18].sVariableValue);
				rBT2RTMall_OG_Sued := STRING_TO_REAL(fbHttp.arrListOfVariabelsOut[19].sVariableValue);
				bBT2PumpenState := DINT_TO_BOOL(STRING_TO_DINT(fbHttp.arrListOfVariabelsOut[20].sVariableValue));
				
				(* ----- Variablen Bauteil 3 ----- *)
				rBT3UmfVorlaufPri := STRING_TO_REAL(fbHttp.arrListOfVariabelsOut[21].sVariableValue);
				rBT3UmfRuecklaufPri := STRING_TO_REAL(fbHttp.arrListOfVariabelsOut[22].sVariableValue);
				rBT3UmfVorlaufSek := STRING_TO_REAL(fbHttp.arrListOfVariabelsOut[23].sVariableValue);
				rBT3UmfRuecklaufSek := STRING_TO_REAL(fbHttp.arrListOfVariabelsOut[24].sVariableValue);
				rBT3RTMall_EG_West := STRING_TO_REAL(fbHttp.arrListOfVariabelsOut[25].sVariableValue);
				rBT3RTMall_OG_West := STRING_TO_REAL(fbHttp.arrListOfVariabelsOut[26].sVariableValue);
				rBT3RTMall_EG_HK31 := STRING_TO_REAL(fbHttp.arrListOfVariabelsOut[27].sVariableValue);
				rBT3RTMall_EG_HK32 := STRING_TO_REAL(fbHttp.arrListOfVariabelsOut[28].sVariableValue);
				rBT3RTMall_OG_K33 := STRING_TO_REAL(fbHttp.arrListOfVariabelsOut[29].sVariableValue);
				rBT3RTMall_OG_K34 := STRING_TO_REAL(fbHttp.arrListOfVariabelsOut[30].sVariableValue);
				rBT3RTMall_OG_Ost := STRING_TO_REAL(fbHttp.arrListOfVariabelsOut[31].sVariableValue);
				rBT3RTMall_EG_Ost := STRING_TO_REAL(fbHttp.arrListOfVariabelsOut[32].sVariableValue);
				rBT3RTMall_EG_HK35 := STRING_TO_REAL(fbHttp.arrListOfVariabelsOut[33].sVariableValue);
				rBT3RTMall_OG_HK37 := STRING_TO_REAL(fbHttp.arrListOfVariabelsOut[34].sVariableValue);
				bBT3PumpenState := DINT_TO_BOOL(STRING_TO_DINT(fbHttp.arrListOfVariabelsOut[35].sVariableValue));
				
				(* ----- Variablen Bauteil 4 ----- *)
				rBT4UmfVorlaufPri := STRING_TO_REAL(fbHttp.arrListOfVariabelsOut[36].sVariableValue);
				rBT4UmfRuecklaufPri := STRING_TO_REAL(fbHttp.arrListOfVariabelsOut[37].sVariableValue);
				rBT4UmfVorlaufSek := STRING_TO_REAL(fbHttp.arrListOfVariabelsOut[38].sVariableValue);
				rBT4UmfRuecklaufSek := STRING_TO_REAL(fbHttp.arrListOfVariabelsOut[39].sVariableValue);
				rBT4RTMall_EG := STRING_TO_REAL(fbHttp.arrListOfVariabelsOut[40].sVariableValue);
				rBT5RTMall_OG := STRING_TO_REAL(fbHttp.arrListOfVariabelsOut[41].sVariableValue);
				rBT6RTMall_OG := STRING_TO_REAL(fbHttp.arrListOfVariabelsOut[42].sVariableValue);
				rBT6RTMall_EG := STRING_TO_REAL(fbHttp.arrListOfVariabelsOut[43].sVariableValue);
				bBT4PumpenState := DINT_TO_BOOL(STRING_TO_DINT(fbHttp.arrListOfVariabelsOut[44].sVariableValue));
				
				(* ----- Wurzelzaehler ----- *)
				lrBT1EM_Counter_kWh := STRING_TO_LREAL(fbHttp.arrListOfVariabelsOut[45].sVariableValue);				
				rBT1EM_Power_kW := STRING_TO_REAL(fbHttp.arrListOfVariabelsOut[46].sVariableValue);
				lrBT2EM_Counter_kWh := STRING_TO_LREAL(fbHttp.arrListOfVariabelsOut[47].sVariableValue);				
				rBT2EM_Power_kW := STRING_TO_REAL(fbHttp.arrListOfVariabelsOut[48].sVariableValue);
				lrBT3EM_Counter_kWh := STRING_TO_LREAL(fbHttp.arrListOfVariabelsOut[49].sVariableValue);				
				rBT3EM_Power_kW := STRING_TO_REAL(fbHttp.arrListOfVariabelsOut[50].sVariableValue);
				lrBT4EM_Counter_kWh := STRING_TO_LREAL(fbHttp.arrListOfVariabelsOut[51].sVariableValue);				
				rBT4EM_Power_kW := STRING_TO_REAL(fbHttp.arrListOfVariabelsOut[52].sVariableValue);
		
		END_IF
			IF FPError.Q THEN iState := 300; END_IF
		
	2://Write Values
	
		// clear array
		FOR byLPArr := 1 TO 100 BY 1 DO
			fbHttp.arrListOfVariables[byLPArr].bIsString := FALSE;
			fbHttp.arrListOfVariables[byLPArr].sVariableName := '';	
			fbHttp.arrListOfVariables[byLPArr].sVariableValue := '';	
		END_FOR
		
		IF fbMonitor.bDissableExtHB THEN byHB := 0; END_IF
		IF fbMonitorBT2.bDissableExtHB THEN byBT2HB := 0; END_IF
		IF fbMonitorBT3.bDissableExtHB THEN byBT3HB := 0; END_IF
		IF fbMonitorBT4.bDissableExtHB THEN byBT4HB := 0; END_IF
	
		fbHttp.bStart := TRUE;	
			fbHttp.bReadRequest := FALSE;
					fbHttp.bWriteRequest := TRUE;
					
		(* ----- Variablen Bauteil 1 ----- *)
		//Watchdog
		fbHttp.arrListOfVariables[1].bIsString := FALSE;
			fbHttp.arrListOfVariables[1].sVariableName := 'DV131';
				fbHttp.arrListOfVariables[1].sVariableValue := REAL_TO_STRING(BYTE_TO_REAL(byHB));		
		//Neuer Sollwert für den Vorlauf für die Regelung
		rNewTargetValue := rNewTargetValue;
		fbHttp.arrListOfVariables[2].bIsString := FALSE;
			fbHttp.arrListOfVariables[2].sVariableName := 'DV133';
				fbHttp.arrListOfVariables[2].sVariableValue := REAL_TO_STRING(rNewTargetValue);	
		
		(* ----- Variablen Bauteil 2 ----- *)
		//Watchdog
		fbHttp.arrListOfVariables[3].bIsString := FALSE;
			fbHttp.arrListOfVariables[3].sVariableName := 'DV231';
				fbHttp.arrListOfVariables[3].sVariableValue := REAL_TO_STRING(BYTE_TO_REAL(byBT2HB));		
		//Neuer Sollwert für den Vorlauf für die Regelung
		rBT2NewTargetValue := rBT2NewTargetValue;
		fbHttp.arrListOfVariables[4].bIsString := FALSE;
			fbHttp.arrListOfVariables[4].sVariableName := 'DV233';
				fbHttp.arrListOfVariables[4].sVariableValue := REAL_TO_STRING(rBT2NewTargetValue);	
		
		(* ----- Variablen Bauteil 3 ----- *)
		//Watchdog
		fbHttp.arrListOfVariables[5].bIsString := FALSE;
			fbHttp.arrListOfVariables[5].sVariableName := 'DV331';
				fbHttp.arrListOfVariables[5].sVariableValue := REAL_TO_STRING(BYTE_TO_REAL(byBT3HB));		
		//Neuer Sollwert für den Vorlauf für die Regelung
		rBT3NewTargetValue := rBT3NewTargetValue;
		fbHttp.arrListOfVariables[6].bIsString := FALSE;
			fbHttp.arrListOfVariables[6].sVariableName := 'DV333';
				fbHttp.arrListOfVariables[6].sVariableValue := REAL_TO_STRING(rBT3NewTargetValue);	
		
		(* ----- Variablen Bauteil 4 ----- *)
		//Watchdog
		fbHttp.arrListOfVariables[7].bIsString := FALSE;
			fbHttp.arrListOfVariables[7].sVariableName := 'DV431';
				fbHttp.arrListOfVariables[7].sVariableValue := REAL_TO_STRING(BYTE_TO_REAL(byBT4HB));		
		//Neuer Sollwert für den Vorlauf für die Regelung
		rBT4NewTargetValue := rBT4NewTargetValue;
		fbHttp.arrListOfVariables[8].bIsString := FALSE;
			fbHttp.arrListOfVariables[8].sVariableName := 'DV433';
				fbHttp.arrListOfVariables[8].sVariableValue := REAL_TO_STRING(rBT4NewTargetValue);	
	
// zusätzliche Variablen laut Markus 23.12.2022 für Heizung schaltern
		// DV132
		x:=9;
		fbHttp.arrListOfVariables[x].bIsString := FALSE;
		fbHttp.arrListOfVariables[x].sVariableName := 'DV132';
		fbHttp.arrListOfVariables[x].sVariableValue := '1';	
		// DV232
		x:=10;
		fbHttp.arrListOfVariables[x].bIsString := FALSE;
		fbHttp.arrListOfVariables[x].sVariableName := 'DV232';
		fbHttp.arrListOfVariables[x].sVariableValue := '1';
		// DV332
		x:=11;
		fbHttp.arrListOfVariables[x].bIsString := FALSE;
		fbHttp.arrListOfVariables[x].sVariableName := 'DV332';
		fbHttp.arrListOfVariables[x].sVariableValue := '1';
		// DV432
		x:=12;
		fbHttp.arrListOfVariables[x].bIsString := FALSE;
		fbHttp.arrListOfVariables[x].sVariableName := 'DV432';
		fbHttp.arrListOfVariables[x].sVariableValue := '1';	
				
		IF FPDone.Q THEN 
			iState := 1; 
				IF NOT fbMonitor.bDissableExtHB THEN byHB := byHB + 1; END_IF
				IF NOT fbMonitorBT2.bDissableExtHB THEN byBT2HB := byBT2HB + 1; END_IF
				IF NOT fbMonitorBT3.bDissableExtHB THEN byBT3HB := byBT3HB + 1; END_IF
				IF NOT fbMonitorBT4.bDissableExtHB THEN byBT4HB := byBT4HB + 1; END_IF
		END_IF
			IF FPError.Q THEN 
				iState := 300; 
					IF NOT fbMonitor.bDissableExtHB THEN byHB := byHB + 1; END_IF
					IF NOT fbMonitorBT2.bDissableExtHB THEN byBT2HB := byBT2HB + 1; END_IF
					IF NOT fbMonitorBT3.bDissableExtHB THEN byBT3HB := byBT3HB + 1; END_IF
					IF NOT fbMonitorBT4.bDissableExtHB THEN byBT4HB := byBT4HB + 1; END_IF
			END_IF
			
		IF byHB > 1 THEN byHB := 0; END_IF
		IF byBT2HB > 1 THEN byBT2HB := 0; END_IF
		IF byBT3HB > 1 THEN byBT3HB := 0; END_IF
		IF byBT4HB > 1 THEN byBT4HB := 0; END_IF
			
	300://Error
		uiErrorCounter := uiErrorCounter + 1;
			iState := 1; 
			
END_CASE

fbHttp(
	bStart:= , 
	bWriteRequest:= , 
	bReadRequest:= , 
	tDelayRequest:= T#10S, 
	sHostname:= '172.24.17.110', 
	arrListOfVariables:= , 
	bValidResult=> , 
	bBusy=> , 
	bError=> , 
	bDone=> , 
	arrListOfVariabelsOut=> , 
	hrErrorCode=> );
	
FPDone(CLK:= fbHttp.bDone, Q=> );
	FPError(CLK:= fbHttp.bError, Q=> );

END_PROGRAM

// ---- FBs/FB_SPOpt_Monitoring_extTime.TcPOU
{attribute 'hide_all_locals'}
FUNCTION_BLOCK FB_SPOpt_Monitoring_extTime
VAR_INPUT PERSISTENT
	bEnable							: BOOL;									//{#lynus.ag#()} //Enable or dissable thsi function
	bDissableHB						: BOOL;									//If this is True, then the Output HB is also dissabled when we have a Error or the Ready Flag from the Backend Service is not OK. If its False the HB is only dissalbed when the Function is not Enables or the HB from the Backend Service is missing
	tChangeHBIn						: TIME := T#70S;						//Delay bettwen the changes from the HB at the Input HB Variable
	tChangeHBOut					: TIME := T#30S;						//Delay bettwen the changes from the HB at the Output HB Variable
END_VAR
VAR_INPUT
	rHeartbeat						: REAL;									//{#lynus.ag#()} //Heartbeat from the Service. NOT OVERRIDE
	rErrorWarning					: REAL;									//{#lynus.ag#()} //Error or Warning from the Service. NOT OVERRIDE
	rSPOptReady						: REAL;									//{#lynus.ag#()} //Setpoint Optimization Service Ready. NOT OVERRIDE
END_VAR
VAR_OUTPUT
	bError							: BOOL;									//Error from this Fuction
	bReadyOut						: BOOL;									//Show if the Service is Read or not
	bDissableExtHB					: BOOL;									//If someone use a external HB with this Flag he can see if the HB, ready or Error Flag from the Backend is set
	bSEnable						: BOOL;									//{#lynus.ag#()} //Enable State of hte function
	rHeartbeatOut					: REAL;									//Heartbeat for the external Service
	diNrOfSPOpt_OUT					: DINT;									//Active Number from Setpoint Optimizer for using on other functions
END_VAR
VAR
	rHBInput_CP						: REAL;									//Variable to compare input HB Variable to set or reset the timer
	fbNumberDevice					: FB_NumberOfDevice;					//Function block to calcualte the number of the Device
	timDissableFunctions			: TON;									//Timer to dissable the Function after Lynus_Standards.Constants_General.tTimeDissableLynusFunctions Days without connection to the Lynus Cloud
	timResetConnectionOnGVL			: TON;									//Timer to try reset the connection Flag on the GVL. (When somebody delete the Connection Function and make only a onlinechange)
	timHBInput						: TON;									//Timer to check the Input HB
	timHBOutput						: TON;									//Timer to set the Output HB
	timReady						: TON;									//Timer to dissable the Ready Flag
	timErrorWarning					: TON;									//Timmer do detect a Error or a Warning
END_VAR

//Creator : Kai Ebensperger
//Company : Lynus AG
//Date : 03.12.2021
//Version : 1.0.0.0

//This is a Function for using with the Setpoin Optimizer on our Backen System.
//So we have the possibility to send the Ready Flag and the HB to the external system we are communicating with in the right intervals.  
//Error evaluation also takes place in this function. Thus, in the event of an error or other event, the Ready flag, the HB or even both can be deactivated and the external system can switch back to classic control. 


(*-------------------------------------------------------------------------------Limits----------------------------------------------------------------------------------------------*)

rHeartbeat := LIMIT(0,rHeartbeat,1);
	rErrorWarning := LIMIT(0,rErrorWarning,2);
		rSPOptReady := LIMIT(0,rSPOptReady,1);
			tChangeHBIn := LIMIT(T#1S,tChangeHBIn,T#1H); // increased this max-Limit due to issues at Cloud-SPO
				tChangeHBOut := LIMIT(T#1S,tChangeHBOut,T#600S);	
	
(*-------------------------------------------------------------Calcualte the number of SP Opttimizer---------------------------------------------------------------*)

fbNumberDevice(
	diActualNumberOfDevices:= Lynus_Standards.GVL_Energy.stNumberOfDevices.diNumberOfSetPointOpt, 
	diMaxNumberOfDevices:= Constants_Energy.diMaxNumberOfSetPointOpt, 
	udiCounterOnlineChange:= TwinCAT_SystemInfoVarList._AppInfo.OnlineChangeCnt, 
	bNumberIsCalculatet=> , 
	bFPNumberIsCalculatet=> , 
	bOnlineChange=> , 
	diNumberForThisDevice=> diNrOfSPOpt_OUT, 
	diNumberOfTotalDevices=> );

//Write new Numer on GVL
IF fbNumberDevice.bFPNumberIsCalculatet THEN
	Lynus_Standards.GVL_Energy.stNumberOfDevices.diNumberOfSetPointOpt := fbNumberDevice.diNumberOfTotalDevices;	
END_IF 

//Delete old Number on GVL
IF fbNumberDevice.bOnlineChange THEN 
	Lynus_Standards.GVL_Energy.stNumberOfDevices.diNumberOfSetPointOpt := diNrOfSPOpt_OUT;
END_IF			
			
(*-------------------------------------------------------------Service from Backend is ready and check the connection to backen for dissabel/enable EMS Function---------------------------------------------------------------*)

//Try to reset the variable for connection on the GVL. When all is normal then the Lynus Mqtt connection function set this variable to true in the next cycle
//When we have no connection to the backend or no HB from the Service then after Lynus_Standards.Constants_General.tTimeDissableLynusFunctions days the EMS is dissabled with all of his functionalities
timResetConnectionOnGVL(IN:= NOT timResetConnectionOnGVL.Q, PT:= T#1H, Q=> , ET=> );
	IF timResetConnectionOnGVL.Q THEN Lynus_Standards.GVL_Communicator.bStateConnectionToEnableFunctions := FALSE; END_IF
		IF NOT Lynus_Standards.GVL_Communicator.bStateConnectionToEnableFunctions OR rHBInput_CP = rHeartbeat THEN timDissableFunctions.IN := TRUE; ELSE timDissableFunctions.IN := FALSE; END_IF  
			timDissableFunctions(IN:= , PT:= Lynus_Standards.Constants_General.tTimeDissableLynusFunctions, Q=> , ET=> );

(*------------------------------------------------------------------Error----------------------------------------------------------------------------*)	

IF Lynus_Standards.GVL_Energy.stNumberOfDevices.diNumberOfSetPointOpt > Constants_Energy.diMaxNumberOfSetPointOpt THEN bError := TRUE; ELSE bError := FALSE; END_IF 
			
(*-----------------------------------------------------------------------------------------------------Logic--------------------------------------------------------------------------------------------------------------*)

bSEnable := bEnable;

//Input HB
timHBInput(IN:= , PT:= tChangeHBIn, Q=> , ET=> );
	IF rHeartbeat <> rHBInput_CP THEN
		timHBInput.IN := FALSE; rHBInput_CP := rHeartbeat;
	ELSE
		timHBInput.IN := TRUE;
	END_IF

//Ready
IF rSPOptReady = 0 THEN timReady.IN := TRUE; ELSE timReady.IN := FALSE; END_IF
	timReady(IN:= , PT:= tChangeHBIn * 2, Q=> , ET=> ); 	
	
//Error and Warning
IF rErrorWarning <> 0 THEN timErrorWarning.IN := TRUE; ELSE timErrorWarning.IN := FALSE; END_IF
	timErrorWarning(IN:= , PT:= tChangeHBIn * 2, Q=> , ET=> );
	
//Set HB Output and Ready Flag
IF rSPOptReady <> 0 AND NOT timReady.Q AND bEnable AND NOT timDissableFunctions.Q AND NOT timErrorWarning.Q THEN bReadyOut := TRUE; END_IF
	IF timReady.Q OR timErrorWarning.Q THEN bReadyOut := FALSE; END_IF

IF (NOT timHBInput.Q AND bDissableHB AND bReadyOut AND NOT timErrorWarning.Q AND NOT timHBOutput.Q AND bEnable AND NOT timDissableFunctions.Q) OR
	(NOT timHBInput.Q AND NOT bDissableHB AND NOT timHBOutput.Q AND bEnable AND NOT timDissableFunctions.Q) THEN
		timHBOutput.IN := TRUE;
ELSE
		timHBOutput.IN := FALSE;
END_IF
	timHBOutput(IN:= , PT:= tChangeHBOut, Q=> , ET=> );
		IF timHBOutput.Q THEN rHeartbeatOut := rHeartbeatOut + 1; END_IF
 			IF rHeartbeatOut > 1 THEN rHeartbeatOut := 0; END_IF

//External HB Flag
IF timHBInput.Q OR (timReady.Q AND bDissableHB) OR (timErrorWarning.Q AND bDissableHB) THEN
	bDissableExtHB := TRUE;
ELSE
	bDissableExtHB := FALSE;
END_IF   
	
//Not Enabled
IF NOT bEnable OR timDissableFunctions.Q OR bError THEN
	bReadyOut := FALSE;
		bDissableExtHB := TRUE;
			rHeartbeatOut := 0;	
END_IF

END_FUNCTION_BLOCK

// ---- POUs/prgPV.TcPOU
PROGRAM prgPV
VAR
	fbSmartLogger_1			: FB_Huawei_SmartLogger;
	fbSmartLogger_2			: FB_Huawei_SmartLogger;
	fbSmartLogger_3			: FB_Huawei_SmartLogger;
	fbPVInt					: FB_PV_Power_Ext_Input;
	fbPVCounter				: FB_EnergyCounter;
	fbPVCounter_1_1			: FB_EnergyCounter;
	fbPVCounter_1_2			: FB_EnergyCounter;
	fbPVCounter_2_1			: FB_EnergyCounter;
	fbPVCounter_2_2			: FB_EnergyCounter;
	fbPVCounter_3_1			: FB_EnergyCounter;
	fbPVCounter_3_2			: FB_EnergyCounter;
	fbPVCounter_3_3			: FB_EnergyCounter;
	fbPVCounter_3_4			: FB_EnergyCounter;
	fbPVCounter_3_5			: FB_EnergyCounter;
	fbPVCounter_3_6			: FB_EnergyCounter;
	lrPowerPV				: LREAL;				//{#lynus.ag#()}
	byErrorWarningPV		: BYTE;					//{#lynus.ag#()}
	
	// extend or reduce amount of PV Inverters
	lrPowerPV_1_1				: LREAL;				//{#lynus.ag#()}
	lrPowerPV_1_2				: LREAL;				//{#lynus.ag#()}
	lrPowerPV_2_1				: LREAL;				//{#lynus.ag#()}
	lrPowerPV_2_2				: LREAL;				//{#lynus.ag#()}
	lrPowerPV_3_1				: LREAL;				//{#lynus.ag#()}
	lrPowerPV_3_2				: LREAL;				//{#lynus.ag#()}
	lrPowerPV_3_3				: LREAL;				//{#lynus.ag#()}
	lrPowerPV_3_4				: LREAL;				//{#lynus.ag#()}
	lrPowerPV_3_5				: LREAL;				//{#lynus.ag#()}
	lrPowerPV_3_6				: LREAL;				//{#lynus.ag#()}
END_VAR
VAR PERSISTENT
	lrCounterPV				: LREAL;				//{#lynus.ag#()}
	lrCounterPV_1_1			: LREAL;				//{#lynus.ag#()}
	lrCounterPV_1_2			: LREAL;				//{#lynus.ag#()}
	lrCounterPV_2_1			: LREAL;				//{#lynus.ag#()}
	lrCounterPV_2_2			: LREAL;				//{#lynus.ag#()}
	lrCounterPV_3_1			: LREAL;				//{#lynus.ag#()}
	lrCounterPV_3_2			: LREAL;				//{#lynus.ag#()}
	lrCounterPV_3_3			: LREAL;				//{#lynus.ag#()}
	lrCounterPV_3_4			: LREAL;				//{#lynus.ag#()}
	lrCounterPV_3_5			: LREAL;				//{#lynus.ag#()}
	lrCounterPV_3_6			: LREAL;				//{#lynus.ag#()}
END_VAR

fbSmartLogger_1(
	bEnable:= TRUE, 
	sIPAdress:= '192.168.34.11', 			// modify IP Adress
	sint_ID_Iverter1 := 12,
	sint_ID_Iverter2 := 13, 
	stDataEMPower_PV=> , 
	stDataEMCounter_PV=> , 
	diNrOfEM_OUT_PV=> );

fbSmartLogger_2(
	bEnable:= TRUE, 
	sIPAdress:= '192.168.34.12', 			// modify IP Adress
	sint_ID_Iverter1 := 12,
	sint_ID_Iverter2 := 13, 
	stDataEMPower_PV=> , 
	stDataEMCounter_PV=> , 
	diNrOfEM_OUT_PV=> );

fbSmartLogger_3(
	bEnable:= TRUE, 
	sIPAdress:= '192.168.34.13', 			// modify IP Adress
	sint_ID_Iverter1 := 11,
	sint_ID_Iverter2 := 72,
	sint_ID_Iverter3 := 73,
	sint_ID_Iverter4 := 74,
	sint_ID_Iverter5 := 75,
	sint_ID_Iverter6 := 76,
	stDataEMPower_PV=> , 
	stDataEMCounter_PV=> , 
	diNrOfEM_OUT_PV=> );
	
// extend or reduce amount of PV Inverters
lrPowerPV_1_1 := fbSmartLogger_1.fbMeter[1].lrPowerTotal / 1000;
lrPowerPV_1_2 := fbSmartLogger_1.fbMeter[2].lrPowerTotal / 1000;
lrPowerPV_2_1 := fbSmartLogger_2.fbMeter[1].lrPowerTotal / 1000;
lrPowerPV_2_2 := fbSmartLogger_2.fbMeter[2].lrPowerTotal / 1000;
lrPowerPV_3_1 := fbSmartLogger_3.fbMeter[1].lrPowerTotal / 1000;
lrPowerPV_3_2 := fbSmartLogger_3.fbMeter[2].lrPowerTotal / 1000;
lrPowerPV_3_3 := fbSmartLogger_3.fbMeter[3].lrPowerTotal / 1000;
lrPowerPV_3_4 := fbSmartLogger_3.fbMeter[4].lrPowerTotal / 1000;
lrPowerPV_3_5 := fbSmartLogger_3.fbMeter[5].lrPowerTotal / 1000;
lrPowerPV_3_6 := fbSmartLogger_3.fbMeter[6].lrPowerTotal / 1000;

	
fbPVInt(
	bEnable:= TRUE, 
	bExtErrorPV := , 
	lrExtPvPower := lrPowerPV_1_1 + lrPowerPV_1_2 + lrPowerPV_2_1 + lrPowerPV_2_2 + lrPowerPV_3_1 + lrPowerPV_3_2 + lrPowerPV_3_3 + lrPowerPV_3_4 + lrPowerPV_3_5 + lrPowerPV_3_6, 
	stDataPv=> , 
	diNrOfPv_OUT=> );
	
lrPowerPV := fbPVInt.stDataPv.lrPower;
	byErrorWarningPV := fbPVInt.stDataPv.byErrorWarning;

// EnergyCounter
fbPVCounter(
	byActiveTariff:= 1, 
	lrPowerInput:= 0 - lrPowerPV, 
	lrTotalCounterEnergy_Consumption=> , 
	lrTotalCounterEnergy_Production=> , 
	lrCounterEnergyT1_Consumption=> , 
	lrCounterEnergyT2_Consumption=> , 
	lrCounterEnergyT1_Production=> , 
	lrCounterEnergyT2_Production=> );
	
IF fbPVCounter.lrTotalCounterEnergy_Production > lrCounterPV THEN  	
	lrCounterPV := fbPVCounter.lrTotalCounterEnergy_Production;
END_IF

fbPVCounter_1_1(
	byActiveTariff:= 1, 
	lrPowerInput:= 0 - lrPowerPV_1_1, 
	lrTotalCounterEnergy_Consumption=> , 
	lrTotalCounterEnergy_Production=> , 
	lrCounterEnergyT1_Consumption=> , 
	lrCounterEnergyT2_Consumption=> , 
	lrCounterEnergyT1_Production=> , 
	lrCounterEnergyT2_Production=> );
	
IF fbPVCounter_1_1.lrTotalCounterEnergy_Production > lrCounterPV_1_1 THEN  	
	lrCounterPV_1_1 := fbPVCounter_1_1.lrTotalCounterEnergy_Production;
END_IF

fbPVCounter_1_2(
	byActiveTariff:= 1, 
	lrPowerInput:= 0 - lrPowerPV_1_2, 
	lrTotalCounterEnergy_Consumption=> , 
	lrTotalCounterEnergy_Production=> , 
	lrCounterEnergyT1_Consumption=> , 
	lrCounterEnergyT2_Consumption=> , 
	lrCounterEnergyT1_Production=> , 
	lrCounterEnergyT2_Production=> );
	
IF fbPVCounter_1_2.lrTotalCounterEnergy_Production > lrCounterPV_1_2 THEN  	
	lrCounterPV_1_2 := fbPVCounter_1_2.lrTotalCounterEnergy_Production;
END_IF

fbPVCounter_2_1(
	byActiveTariff:= 1, 
	lrPowerInput:= 0 - lrPowerPV_2_1, 
	lrTotalCounterEnergy_Consumption=> , 
	lrTotalCounterEnergy_Production=> , 
	lrCounterEnergyT1_Consumption=> , 
	lrCounterEnergyT2_Consumption=> , 
	lrCounterEnergyT1_Production=> , 
	lrCounterEnergyT2_Production=> );
	
IF fbPVCounter_2_1.lrTotalCounterEnergy_Production > lrCounterPV_2_1 THEN  	
	lrCounterPV_2_1 := fbPVCounter_2_1.lrTotalCounterEnergy_Production;
END_IF

fbPVCounter_2_2(
	byActiveTariff:= 1, 
	lrPowerInput:= 0 - lrPowerPV_2_2, 
	lrTotalCounterEnergy_Consumption=> , 
	lrTotalCounterEnergy_Production=> , 
	lrCounterEnergyT1_Consumption=> , 
	lrCounterEnergyT2_Consumption=> , 
	lrCounterEnergyT1_Production=> , 
	lrCounterEnergyT2_Production=> );
	
IF fbPVCounter_2_2.lrTotalCounterEnergy_Production > lrCounterPV_2_2 THEN  	
	lrCounterPV_2_2 := fbPVCounter_2_2.lrTotalCounterEnergy_Production;
END_IF

fbPVCounter_3_1(
	byActiveTariff:= 1, 
	lrPowerInput:= 0 - lrPowerPV_3_1, 
	lrTotalCounterEnergy_Consumption=> , 
	lrTotalCounterEnergy_Production=> , 
	lrCounterEnergyT1_Consumption=> , 
	lrCounterEnergyT2_Consumption=> , 
	lrCounterEnergyT1_Production=> , 
	lrCounterEnergyT2_Production=> );
	
IF fbPVCounter_3_1.lrTotalCounterEnergy_Production > lrCounterPV_3_1 THEN  	
	lrCounterPV_3_1 := fbPVCounter_3_1.lrTotalCounterEnergy_Production;
END_IF

fbPVCounter_3_2(
	byActiveTariff:= 1, 
	lrPowerInput:= 0 - lrPowerPV_3_2, 
	lrTotalCounterEnergy_Consumption=> , 
	lrTotalCounterEnergy_Production=> , 
	lrCounterEnergyT1_Consumption=> , 
	lrCounterEnergyT2_Consumption=> , 
	lrCounterEnergyT1_Production=> , 
	lrCounterEnergyT2_Production=> );
	
IF fbPVCounter_3_2.lrTotalCounterEnergy_Production > lrCounterPV_3_2 THEN  	
	lrCounterPV_3_2 := fbPVCounter_3_2.lrTotalCounterEnergy_Production;
END_IF

fbPVCounter_3_3(
	byActiveTariff:= 1, 
	lrPowerInput:= 0 - lrPowerPV_3_3, 
	lrTotalCounterEnergy_Consumption=> , 
	lrTotalCounterEnergy_Production=> , 
	lrCounterEnergyT1_Consumption=> , 
	lrCounterEnergyT2_Consumption=> , 
	lrCounterEnergyT1_Production=> , 
	lrCounterEnergyT2_Production=> );
	
IF fbPVCounter_3_3.lrTotalCounterEnergy_Production > lrCounterPV_3_3 THEN  	
	lrCounterPV_3_3 := fbPVCounter_3_3.lrTotalCounterEnergy_Production;
END_IF

fbPVCounter_3_4(
	byActiveTariff:= 1, 
	lrPowerInput:= 0 - lrPowerPV_3_4, 
	lrTotalCounterEnergy_Consumption=> , 
	lrTotalCounterEnergy_Production=> , 
	lrCounterEnergyT1_Consumption=> , 
	lrCounterEnergyT2_Consumption=> , 
	lrCounterEnergyT1_Production=> , 
	lrCounterEnergyT2_Production=> );
	
IF fbPVCounter_3_4.lrTotalCounterEnergy_Production > lrCounterPV_3_4 THEN  	
	lrCounterPV_3_4 := fbPVCounter_3_4.lrTotalCounterEnergy_Production;
END_IF

fbPVCounter_3_5(
	byActiveTariff:= 1, 
	lrPowerInput:= 0 - lrPowerPV_3_5, 
	lrTotalCounterEnergy_Consumption=> , 
	lrTotalCounterEnergy_Production=> , 
	lrCounterEnergyT1_Consumption=> , 
	lrCounterEnergyT2_Consumption=> , 
	lrCounterEnergyT1_Production=> , 
	lrCounterEnergyT2_Production=> );
	
IF fbPVCounter_3_5.lrTotalCounterEnergy_Production > lrCounterPV_3_5 THEN  	
	lrCounterPV_3_5 := fbPVCounter_3_5.lrTotalCounterEnergy_Production;
END_IF

fbPVCounter_3_6(
	byActiveTariff:= 1, 
	lrPowerInput:= 0 - lrPowerPV_3_6, 
	lrTotalCounterEnergy_Consumption=> , 
	lrTotalCounterEnergy_Production=> , 
	lrCounterEnergyT1_Consumption=> , 
	lrCounterEnergyT2_Consumption=> , 
	lrCounterEnergyT1_Production=> , 
	lrCounterEnergyT2_Production=> );
	
IF fbPVCounter_3_6.lrTotalCounterEnergy_Production > lrCounterPV_3_6 THEN  	
	lrCounterPV_3_6 := fbPVCounter_3_6.lrTotalCounterEnergy_Production;
END_IF

END_PROGRAM

// ---- POUs/prgLynus.TcPOU
PROGRAM prgLynus
VAR
	fbRW1		: FB_ReadWrite_V2;
END_VAR

fbRW1(
	eUploadType:= eSelectDataUploadType.e_Change_Intervall5min , 
	bBusy=> , 
	bError=> , 
	udiErrorCodeOut=> , 
	eErrorReadWrite_Out=> );

END_PROGRAM
